(* CODESYS project Networkvariables.recver.project
   Description: This example demonstrates how to share a variable within a network. One application is sending the variable and the other one receives it.
   Title: Network Variables
   Version: 1.0.0.0
   Company: 3S - Smart Software Solutions GmbH

Project tree, tasks and I/O mapping:
  Receiver : Changsha-Cyber-MI-linux, Changsha Cyber-MI Co., Ltd., version 3.5.10.40
    application App_Receive
      libraries: Standard, * (System)
      task Task (cyclic, interval t#20ms, priority 1) calls Main_Receive
      declarations NVL
      program Main_Receive [ST]
    SoftMotion General Axis Pool
*)

// Receiver/App_Receive/NVL
//This gobal variable list is received via the network.
//Sender: Imported from file 'D:\Data.gvl'
//Protocol: UDP

{attribute 'qualified_only'}
VAR_GLOBAL
	iglobvar:INT; 
	bGlobVar01:BOOL;
	uGlobVar03:UINT;
	uGlobVar04:UINT;
	uGlobVar05:UINT;
END_VAR

// Receiver/App_Receive/Main_Receive
PROGRAM Main_Receive
VAR
	ivarLocal : INT;
	
	RxDiag : NetVarUdp.NetVarUDPDiagStruct;
END_VAR

ivarLocal := nvl.iglobvar;

(* Diagnostic *)
RxDiag := NetVar_App_Receive_GVL.NetVarRxDiag_UDP[0];

END_PROGRAM
